(* PLC project graf, TNI-Software ControlBuild 4.00 *)
(* stored: creationDateTime 2018-09-17T16:16:55-01:00 *)

CONFIGURATION graf
  VAR_GLOBAL
    simuperiod : REAL := 50000.0;
    taskname : STRING(50) := 'graf.exe';
    allowpreconditions : BOOL := true;
    allowpostconditions : BOOL := true;
  END_VAR
END_CONFIGURATION
